// TIA Portal V16 export
// export: Created 2021-07-12T14:47:18.226577Z, ExportSetting WithDefaults, DisplayName Totally Integrated Automation Portal, DisplayVersion V16, DisplayName TIA Portal Version Control Interface, DisplayVersion V16, DisplayName TIA Portal Openness, DisplayVersion V16, DisplayName STEP 7 Professional, DisplayVersion V16, DisplayName STEP 7 Safety, DisplayVersion V16, DisplayName WinCC Professional, DisplayVersion V16
TYPE "LSimaHydTO_typeStatusActor"
TITLE = LSimaHydTO_typeStatusActor
// Indicates the status of actor data
// stored: IsFailsafeCompliant false
   STRUCT
      SetPoint : LReal := 0.0;   // Manipulated variable
      AddSetPoint : LReal := 0.0;   // Additional setpoint
      QOutputValue : LReal := 0.0;   // Output value in relation to Q-output [%]
      Enabled : Bool;   // Output is enabled
      ValveForward : Bool := FALSE;   // Control bit for positive direction
      ValveBackward : Bool := FALSE;   // Control bit for negative direction
   END_STRUCT;
END_TYPE
